// TIA Portal V18 export
FUNCTION "Verify_Settings" : Void   // FC21, LAD
{ S7_Optimized_Access := 'TRUE' }
// Written BY Kristopher Gimenez February 9th, 2023
// This block is used to check the settings are within limits and adjust as needed
// stored: AutoNumber false, SetENOAutomatically false
BEGIN

REGION Network 1: Alpha Values
   // All alpha filter values between 0-1
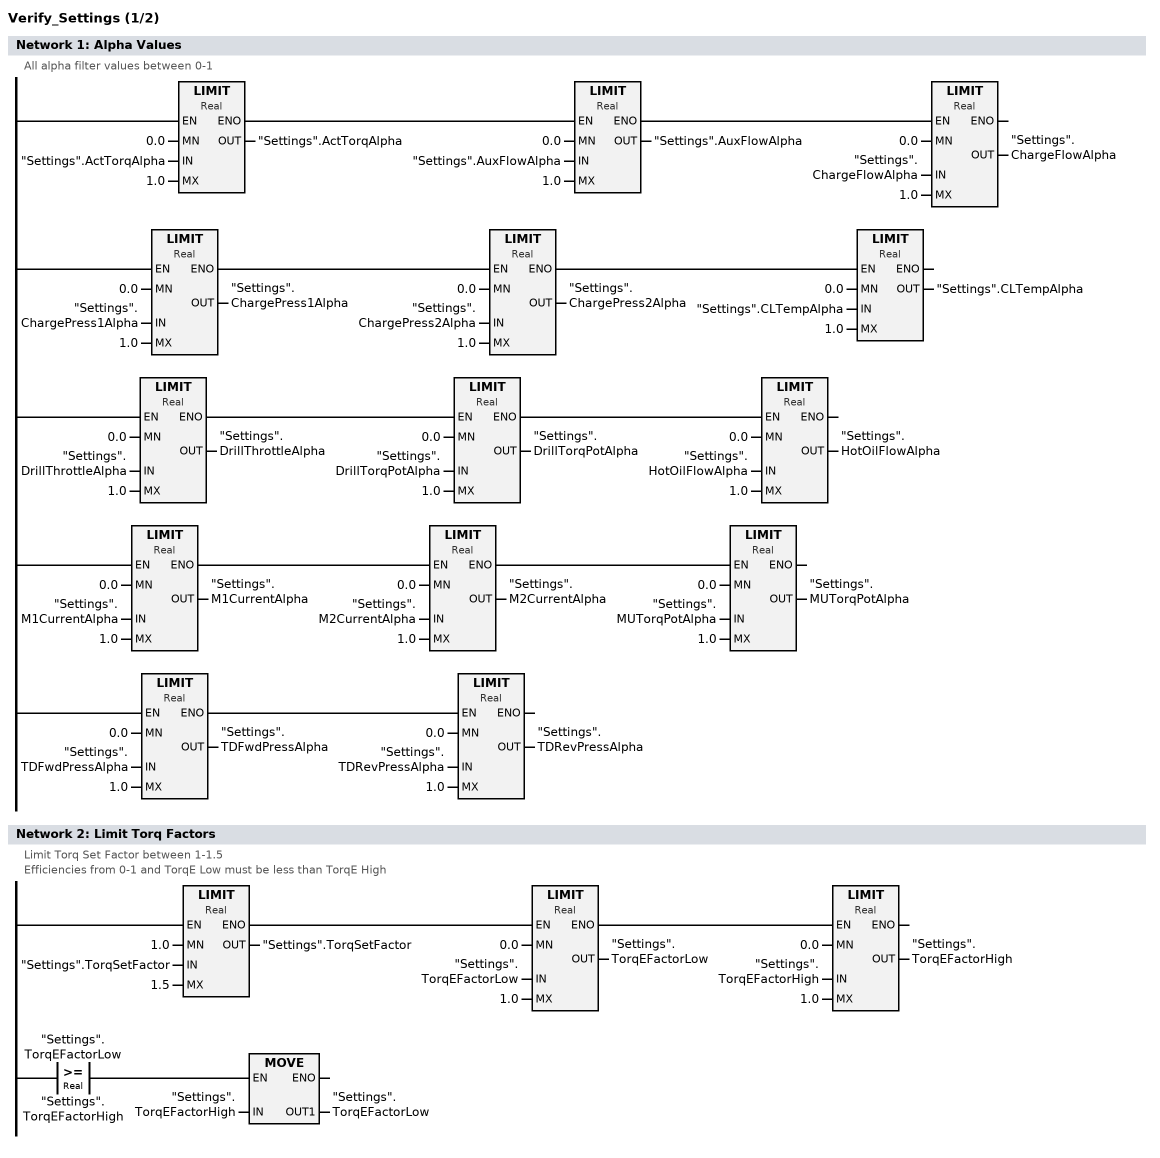
   RUNG wire#powerrail
      { S7_Templates := "value_type := Real" } Limit(mn := 0.0, in := "Settings".ActTorqAlpha, mx := 1.0, out => "Settings".ActTorqAlpha)
      { S7_Templates := "value_type := Real" } Limit(mn := 0.0, in := "Settings".AuxFlowAlpha, mx := 1.0, out => "Settings".AuxFlowAlpha)
      { S7_Templates := "value_type := Real" } Limit(mn := 0.0, in := "Settings".ChargeFlowAlpha, mx := 1.0, out => "Settings".ChargeFlowAlpha)
   END_RUNG
   RUNG wire#powerrail
      { S7_Templates := "value_type := Real" } Limit(mn := 0.0, in := "Settings".ChargePress1Alpha, mx := 1.0, out => "Settings".ChargePress1Alpha)
      { S7_Templates := "value_type := Real" } Limit(mn := 0.0, in := "Settings".ChargePress2Alpha, mx := 1.0, out => "Settings".ChargePress2Alpha)
      { S7_Templates := "value_type := Real" } Limit(mn := 0.0, in := "Settings".CLTempAlpha, mx := 1.0, out => "Settings".CLTempAlpha)
   END_RUNG
   RUNG wire#powerrail
      { S7_Templates := "value_type := Real" } Limit(mn := 0.0, in := "Settings".DrillThrottleAlpha, mx := 1.0, out => "Settings".DrillThrottleAlpha)
      { S7_Templates := "value_type := Real" } Limit(mn := 0.0, in := "Settings".DrillTorqPotAlpha, mx := 1.0, out => "Settings".DrillTorqPotAlpha)
      { S7_Templates := "value_type := Real" } Limit(mn := 0.0, in := "Settings".HotOilFlowAlpha, mx := 1.0, out => "Settings".HotOilFlowAlpha)
   END_RUNG
   RUNG wire#powerrail
      { S7_Templates := "value_type := Real" } Limit(mn := 0.0, in := "Settings".M1CurrentAlpha, mx := 1.0, out => "Settings".M1CurrentAlpha)
      { S7_Templates := "value_type := Real" } Limit(mn := 0.0, in := "Settings".M2CurrentAlpha, mx := 1.0, out => "Settings".M2CurrentAlpha)
      { S7_Templates := "value_type := Real" } Limit(mn := 0.0, in := "Settings".MUTorqPotAlpha, mx := 1.0, out => "Settings".MUTorqPotAlpha)
   END_RUNG
   RUNG wire#powerrail
      { S7_Templates := "value_type := Real" } Limit(mn := 0.0, in := "Settings".TDFwdPressAlpha, mx := 1.0, out => "Settings".TDFwdPressAlpha)
      { S7_Templates := "value_type := Real" } Limit(mn := 0.0, in := "Settings".TDRevPressAlpha, mx := 1.0, out => "Settings".TDRevPressAlpha)
   END_RUNG
   // the same network as SCL:
   "Settings".ActTorqAlpha := LIMIT(MN := 0.0, IN := "Settings".ActTorqAlpha, MX := 1.0);
   "Settings".AuxFlowAlpha := LIMIT(MN := 0.0, IN := "Settings".AuxFlowAlpha, MX := 1.0);
   "Settings".ChargeFlowAlpha := LIMIT(MN := 0.0, IN := "Settings".ChargeFlowAlpha, MX := 1.0);
   "Settings".ChargePress1Alpha := LIMIT(MN := 0.0, IN := "Settings".ChargePress1Alpha, MX := 1.0);
   "Settings".ChargePress2Alpha := LIMIT(MN := 0.0, IN := "Settings".ChargePress2Alpha, MX := 1.0);
   "Settings".CLTempAlpha := LIMIT(MN := 0.0, IN := "Settings".CLTempAlpha, MX := 1.0);
   "Settings".DrillThrottleAlpha := LIMIT(MN := 0.0, IN := "Settings".DrillThrottleAlpha, MX := 1.0);
   "Settings".DrillTorqPotAlpha := LIMIT(MN := 0.0, IN := "Settings".DrillTorqPotAlpha, MX := 1.0);
   "Settings".HotOilFlowAlpha := LIMIT(MN := 0.0, IN := "Settings".HotOilFlowAlpha, MX := 1.0);
   "Settings".M1CurrentAlpha := LIMIT(MN := 0.0, IN := "Settings".M1CurrentAlpha, MX := 1.0);
   "Settings".M2CurrentAlpha := LIMIT(MN := 0.0, IN := "Settings".M2CurrentAlpha, MX := 1.0);
   "Settings".MUTorqPotAlpha := LIMIT(MN := 0.0, IN := "Settings".MUTorqPotAlpha, MX := 1.0);
   "Settings".TDFwdPressAlpha := LIMIT(MN := 0.0, IN := "Settings".TDFwdPressAlpha, MX := 1.0);
   "Settings".TDRevPressAlpha := LIMIT(MN := 0.0, IN := "Settings".TDRevPressAlpha, MX := 1.0);
END_REGION

REGION Network 2: Limit Torq Factors
   // Limit Torq Set Factor between 1-1.5
   // Efficiencies from 0-1 and TorqE Low must be less than TorqE High
   RUNG wire#powerrail
      { S7_Templates := "value_type := Real" } Limit(mn := 1.0, in := "Settings".TorqSetFactor, mx := 1.5, out => "Settings".TorqSetFactor)
      { S7_Templates := "value_type := Real" } Limit(mn := 0.0, in := "Settings".TorqEFactorLow, mx := 1.0, out => "Settings".TorqEFactorLow)
      { S7_Templates := "value_type := Real" } Limit(mn := 0.0, in := "Settings".TorqEFactorHigh, mx := 1.0, out => "Settings".TorqEFactorHigh)
   END_RUNG
   RUNG wire#powerrail
      { S7_Templates := "SrcType := Real" } GE_Contact(in1 := "Settings".TorqEFactorLow, in2 := "Settings".TorqEFactorHigh)
      Move(in := "Settings".TorqEFactorHigh, out1 => "Settings".TorqEFactorLow)
   END_RUNG
   // the same network as SCL:
   "Settings".TorqSetFactor := LIMIT(MN := 1.0, IN := "Settings".TorqSetFactor, MX := 1.5);
   "Settings".TorqEFactorLow := LIMIT(MN := 0.0, IN := "Settings".TorqEFactorLow, MX := 1.0);
   "Settings".TorqEFactorHigh := LIMIT(MN := 0.0, IN := "Settings".TorqEFactorHigh, MX := 1.0);
   IF "Settings".TorqEFactorLow >= "Settings".TorqEFactorHigh THEN
       "Settings".TorqEFactorLow := "Settings".TorqEFactorHigh;
   END_IF;
END_REGION

REGION Network 3: Verify BO Setting
   // BO Spin Factor from 1-2
   // Shift RPM from 1 to Speed limit
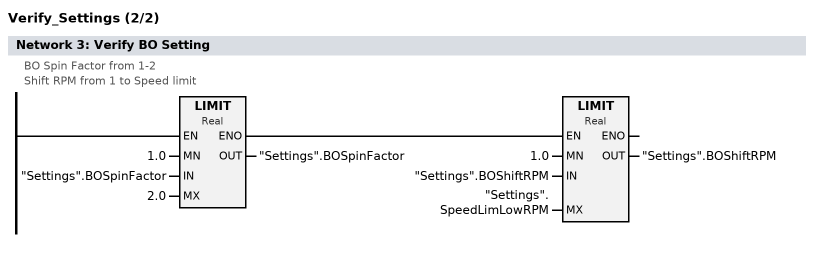
   RUNG wire#powerrail
      { S7_Templates := "value_type := Real" } Limit(mn := 1.0, in := "Settings".BOSpinFactor, mx := 2.0, out => "Settings".BOSpinFactor)
      { S7_Templates := "value_type := Real" } Limit(mn := 1.0, in := "Settings".BOShiftRPM, mx := "Settings".SpeedLimLowRPM, out => "Settings".BOShiftRPM)
   END_RUNG
   // the same network as SCL:
   "Settings".BOSpinFactor := LIMIT(MN := 1.0, IN := "Settings".BOSpinFactor, MX := 2.0);
   "Settings".BOShiftRPM := LIMIT(MN := 1.0, IN := "Settings".BOShiftRPM, MX := "Settings".SpeedLimLowRPM);
END_REGION
END_FUNCTION
